# EPICS substitutions: epics/m-epics-eemcu/eemcuApp/Db/Sim8-extra-m6.substitutions
file "eemcu-extra.template"
{
pattern
{P,      M,    R,   PORT, ADDR, PREC, HOMEPROC}
{IOC:,   m6, m6-,   MCU1,    6, 3,    3}
}
